# EPICS autosave request: motorApp/Db/profileMoveControllerXPS_settings.req
$(P)$(R)TrajectoryFile
$(P)$(R)GroupName
